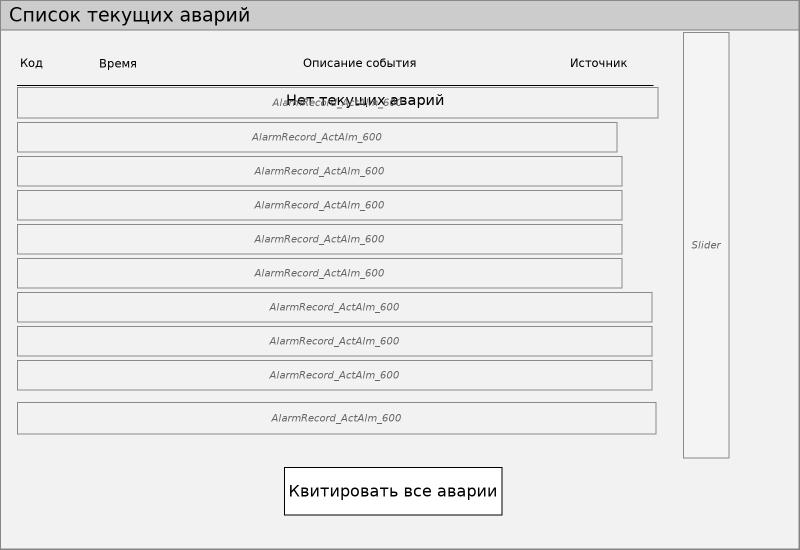
VISUALIZATION Current_Alarms_800x550  // 800x550
    Rectangle (0,0 800x550)
    Frame (17,122 600x30)
        shows AlarmRecord_ActAlm_600(AlarmRecord := PRG_Alarms_Core.HMI_ActiveAlarms[2])
    Frame (17,156 605x30)
        shows AlarmRecord_ActAlm_600(AlarmRecord := PRG_Alarms_Core.HMI_ActiveAlarms[3])
    Frame (17,190 605x30)
        shows AlarmRecord_ActAlm_600(AlarmRecord := PRG_Alarms_Core.HMI_ActiveAlarms[4])
    Frame (17,224 605x30)
        shows AlarmRecord_ActAlm_600(AlarmRecord := PRG_Alarms_Core.HMI_ActiveAlarms[5])
    Frame (17,258 605x30)
        shows AlarmRecord_ActAlm_600(AlarmRecord := PRG_Alarms_Core.HMI_ActiveAlarms[6])
    Frame (17,292 635x30)
        shows AlarmRecord_ActAlm_600(AlarmRecord := PRG_Alarms_Core.HMI_ActiveAlarms[7])
    Frame (17,326 635x30)
        shows AlarmRecord_ActAlm_600(AlarmRecord := PRG_Alarms_Core.HMI_ActiveAlarms[8])
    Frame (17,360 635x30)
        shows AlarmRecord_ActAlm_600(AlarmRecord := PRG_Alarms_Core.HMI_ActiveAlarms[9])
    Frame (17,402 639x32)
        shows AlarmRecord_ActAlm_600(AlarmRecord := PRG_Alarms_Core.HMI_ActiveAlarms[10])
    Label (250,85 231x30), "Нет текущих аварий", invisible if: PRG_Alarms_Core.HMI_ActiveAlarms[1].isActive
    Frame (17,87 641x31)
        shows AlarmRecord_ActAlm_600(AlarmRecord := PRG_Alarms_Core.HMI_ActiveAlarms[1])
    Rectangle (0,0 800x30), "Список текущих аварий"
    Slider (683,32 46x426), variable: PRG_Alarms_Core.HMI_CurShiftAA, scale 0..1000
    Label (17,48 37x30), "Код"
    Label (300,48 216x30), "Описание события"
    Label (567,48 77x30), "Источник"
    Label (92,54 52x19), "Время"
    Line (17,85) (653,85)
    RoundedRectangle (284,467 218x48), "Квитировать все аварии"
        tap LibAlarm.bLocalQuitAllAlarms
END_VISUALIZATION

(* stored: Version 1.1.0.1, ProductVersion 3.1.4024.9
   Visu Current_Alarms_800x550: Id {216bf934-fa18-4df6-9511-3aad321675c2} *)
